// TIA Portal V16 export
// export: Created 2023-03-29T11:03:47.9785321Z, ExportSetting WithDefaults, DisplayName Totally Integrated Automation Portal, DisplayVersion V16 Update 6, DisplayName TIA Portal Version Control Interface, DisplayVersion V16 Update 2, DisplayName TIA Portal Openness, DisplayVersion V16 Update 6, DisplayName STEP 7 Professional, DisplayVersion V16 Update 6, DisplayName STEP 7 Safety, DisplayVersion V16, DisplayName WinCC Advanced, DisplayVersion V16 Update 6
TYPE "typeDataInverter_Byte"
// stored: IsFailsafeCompliant false
   STRUCT
      typeDataInverter_byte : Array[0..0] of Byte;   // Typ dane byte, falownik
   END_STRUCT;
END_TYPE
